// TIA Portal V19 export
TYPE "SiemensDataType"
   STRUCT
      Test1 : Bool;
      Test2 : Bool;
      Test3 : Bool;
      Test4 : Bool;
      Test5 : Bool;
      Test6 : Bool;
      Test7 : Bool;
   END_STRUCT;
END_TYPE
